REGION Network 109: Step[730] : Z1, Z2 aviod Pos move
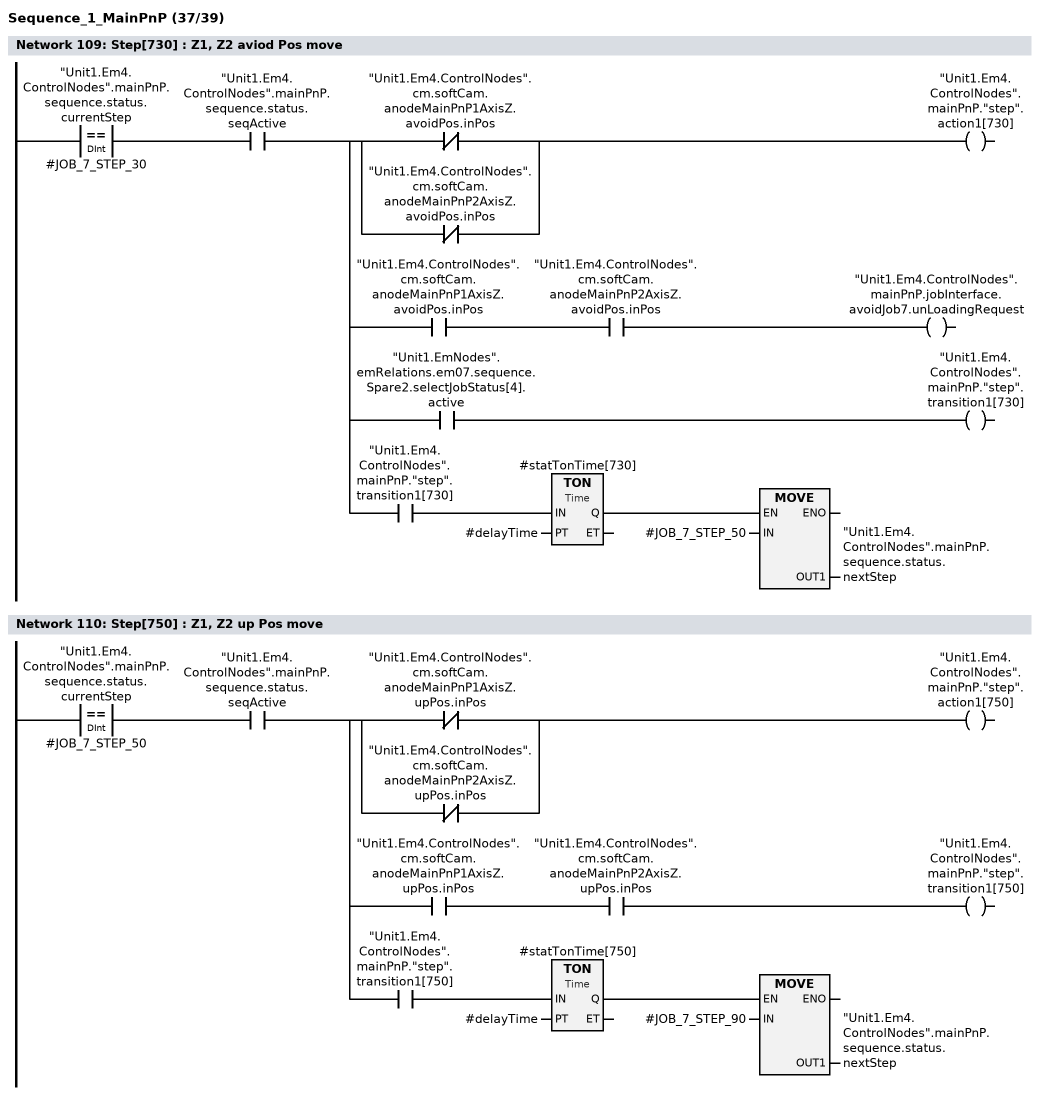
   RUNG wire#powerrail
      { S7_Templates := "SrcType := DInt" } EQ_Contact(in1 := "Unit1.Em4.ControlNodes".mainPnP.sequence.status.currentStep, in2 := #JOB_7_STEP_30)
      Contact( "Unit1.Em4.ControlNodes".mainPnP.sequence.status.seqActive )
      wire#w1
      I_Contact( "Unit1.Em4.ControlNodes".cm.softCam.anodeMainPnP1AxisZ.avoidPos.inPos )
      wire#w2
      Coil( "Unit1.Em4.ControlNodes".mainPnP."step".action1[730] )
   END_RUNG
   RUNG wire#w1
      I_Contact( "Unit1.Em4.ControlNodes".cm.softCam.anodeMainPnP2AxisZ.avoidPos.inPos )
   END_RUNG wire#w2
   RUNG wire#w1
      Contact( "Unit1.Em4.ControlNodes".cm.softCam.anodeMainPnP1AxisZ.avoidPos.inPos )
      Contact( "Unit1.Em4.ControlNodes".cm.softCam.anodeMainPnP2AxisZ.avoidPos.inPos )
      Coil( "Unit1.Em4.ControlNodes".mainPnP.jobInterface.avoidJob7.unLoadingRequest )
   END_RUNG
   RUNG wire#w1
      Contact( "Unit1.EmNodes".emRelations.em07.sequence.Spare2.selectJobStatus[4].active )
      Coil( "Unit1.Em4.ControlNodes".mainPnP."step".transition1[730] )
   END_RUNG
   RUNG wire#w1
      Contact( "Unit1.Em4.ControlNodes".mainPnP."step".transition1[730] )
      { S7_Templates := "time_type := Time" } #statTonTime[730].TON(pt := #delayTime, et =>)
      Move(in := #JOB_7_STEP_50, out1 => "Unit1.Em4.ControlNodes".mainPnP.sequence.status.nextStep)
   END_RUNG
   // the same network as SCL:
   #_w1 := ("Unit1.Em4.ControlNodes".mainPnP.sequence.status.currentStep = #JOB_7_STEP_30) AND "Unit1.Em4.ControlNodes".mainPnP.sequence.status.seqActive;
   "Unit1.Em4.ControlNodes".mainPnP."step".action1[730] := #_w1 AND (NOT "Unit1.Em4.ControlNodes".cm.softCam.anodeMainPnP1AxisZ.avoidPos.inPos OR NOT "Unit1.Em4.ControlNodes".cm.softCam.anodeMainPnP2AxisZ.avoidPos.inPos);
   "Unit1.Em4.ControlNodes".mainPnP.jobInterface.avoidJob7.unLoadingRequest := #_w1 AND "Unit1.Em4.ControlNodes".cm.softCam.anodeMainPnP1AxisZ.avoidPos.inPos AND "Unit1.Em4.ControlNodes".cm.softCam.anodeMainPnP2AxisZ.avoidPos.inPos;
   "Unit1.Em4.ControlNodes".mainPnP."step".transition1[730] := #_w1 AND "Unit1.EmNodes".emRelations.em07.sequence.Spare2.selectJobStatus[4].active;
   #statTonTime[730].TON(IN := #_w1 AND "Unit1.Em4.ControlNodes".mainPnP."step".transition1[730],
                         PT := #delayTime);
   IF #statTonTime[730].Q THEN
       "Unit1.Em4.ControlNodes".mainPnP.sequence.status.nextStep := #JOB_7_STEP_50;
   END_IF;
END_REGION

REGION Network 110: Step[750] : Z1, Z2 up Pos move
   RUNG wire#powerrail
      { S7_Templates := "SrcType := DInt" } EQ_Contact(in1 := "Unit1.Em4.ControlNodes".mainPnP.sequence.status.currentStep, in2 := #JOB_7_STEP_50)
      Contact( "Unit1.Em4.ControlNodes".mainPnP.sequence.status.seqActive )
      wire#w1
      I_Contact( "Unit1.Em4.ControlNodes".cm.softCam.anodeMainPnP1AxisZ.upPos.inPos )
      wire#w2
      Coil( "Unit1.Em4.ControlNodes".mainPnP."step".action1[750] )
   END_RUNG
   RUNG wire#w1
      I_Contact( "Unit1.Em4.ControlNodes".cm.softCam.anodeMainPnP2AxisZ.upPos.inPos )
   END_RUNG wire#w2
   RUNG wire#w1
      Contact( "Unit1.Em4.ControlNodes".cm.softCam.anodeMainPnP1AxisZ.upPos.inPos )
      Contact( "Unit1.Em4.ControlNodes".cm.softCam.anodeMainPnP2AxisZ.upPos.inPos )
      Coil( "Unit1.Em4.ControlNodes".mainPnP."step".transition1[750] )
   END_RUNG
   RUNG wire#w1
      Contact( "Unit1.Em4.ControlNodes".mainPnP."step".transition1[750] )
      { S7_Templates := "time_type := Time" } #statTonTime[750].TON(pt := #delayTime, et =>)
      Move(in := #JOB_7_STEP_90, out1 => "Unit1.Em4.ControlNodes".mainPnP.sequence.status.nextStep)
   END_RUNG
   // the same network as SCL:
   #_w1 := ("Unit1.Em4.ControlNodes".mainPnP.sequence.status.currentStep = #JOB_7_STEP_50) AND "Unit1.Em4.ControlNodes".mainPnP.sequence.status.seqActive;
   "Unit1.Em4.ControlNodes".mainPnP."step".action1[750] := #_w1 AND (NOT "Unit1.Em4.ControlNodes".cm.softCam.anodeMainPnP1AxisZ.upPos.inPos OR NOT "Unit1.Em4.ControlNodes".cm.softCam.anodeMainPnP2AxisZ.upPos.inPos);
   "Unit1.Em4.ControlNodes".mainPnP."step".transition1[750] := #_w1 AND "Unit1.Em4.ControlNodes".cm.softCam.anodeMainPnP1AxisZ.upPos.inPos AND "Unit1.Em4.ControlNodes".cm.softCam.anodeMainPnP2AxisZ.upPos.inPos;
   #statTonTime[750].TON(IN := #_w1 AND "Unit1.Em4.ControlNodes".mainPnP."step".transition1[750],
                         PT := #delayTime);
   IF #statTonTime[750].Q THEN
       "Unit1.Em4.ControlNodes".mainPnP.sequence.status.nextStep := #JOB_7_STEP_90;
   END_IF;
END_REGION

REGION Network 111: Step[790] : JOB[7] Condition
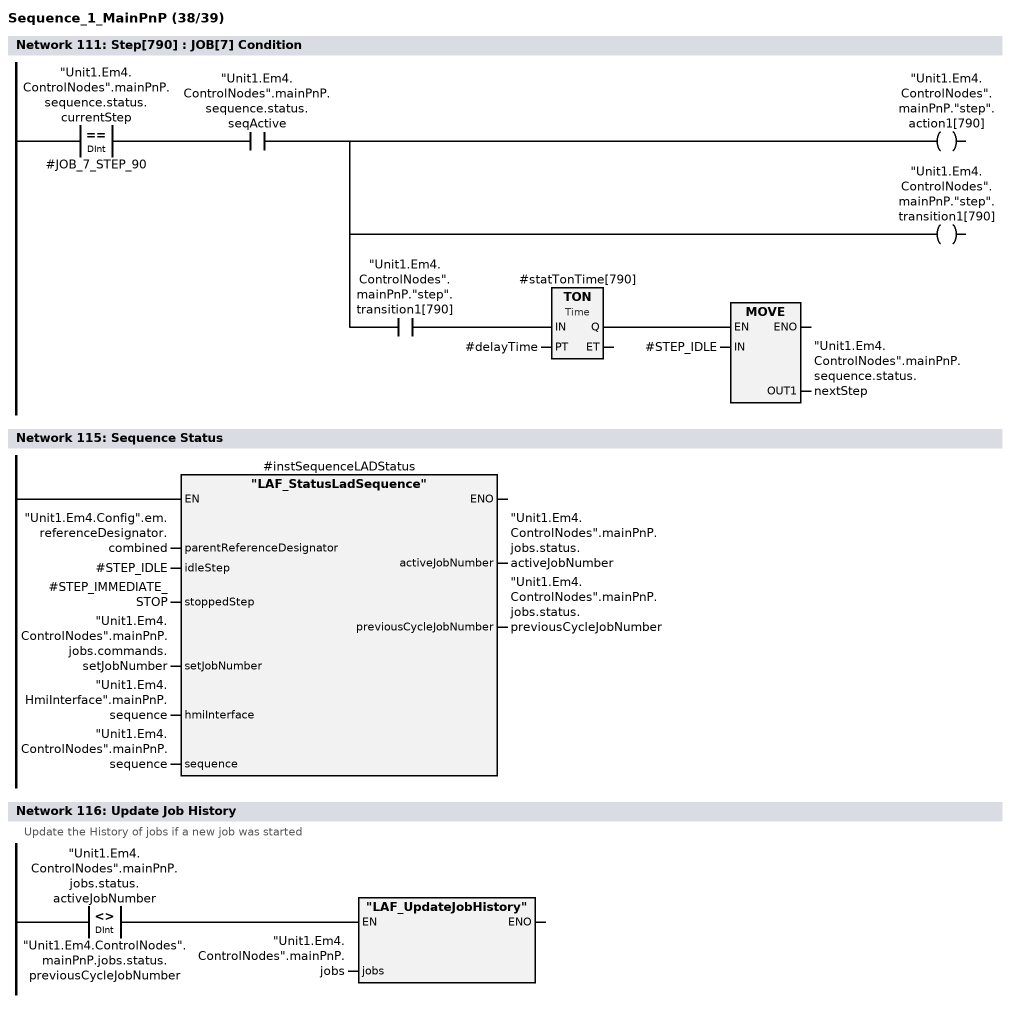
   RUNG wire#powerrail
      { S7_Templates := "SrcType := DInt" } EQ_Contact(in1 := "Unit1.Em4.ControlNodes".mainPnP.sequence.status.currentStep, in2 := #JOB_7_STEP_90)
      Contact( "Unit1.Em4.ControlNodes".mainPnP.sequence.status.seqActive )
      wire#w1
      Coil( "Unit1.Em4.ControlNodes".mainPnP."step".action1[790] )
   END_RUNG
   RUNG wire#w1
      Coil( "Unit1.Em4.ControlNodes".mainPnP."step".transition1[790] )
   END_RUNG
   RUNG wire#w1
      Contact( "Unit1.Em4.ControlNodes".mainPnP."step".transition1[790] )
      { S7_Templates := "time_type := Time" } #statTonTime[790].TON(pt := #delayTime, et =>)
      Move(in := #STEP_IDLE, out1 => "Unit1.Em4.ControlNodes".mainPnP.sequence.status.nextStep)
   END_RUNG
   // the same network as SCL:
   "Unit1.Em4.ControlNodes".mainPnP."step".action1[790] := ("Unit1.Em4.ControlNodes".mainPnP.sequence.status.currentStep = #JOB_7_STEP_90) AND "Unit1.Em4.ControlNodes".mainPnP.sequence.status.seqActive;
   "Unit1.Em4.ControlNodes".mainPnP."step".transition1[790] := ("Unit1.Em4.ControlNodes".mainPnP.sequence.status.currentStep = #JOB_7_STEP_90) AND "Unit1.Em4.ControlNodes".mainPnP.sequence.status.seqActive;
   #statTonTime[790].TON(IN := ("Unit1.Em4.ControlNodes".mainPnP.sequence.status.currentStep = #JOB_7_STEP_90) AND "Unit1.Em4.ControlNodes".mainPnP.sequence.status.seqActive AND "Unit1.Em4.ControlNodes".mainPnP."step".transition1[790],
                         PT := #delayTime);
   IF #statTonTime[790].Q THEN
       "Unit1.Em4.ControlNodes".mainPnP.sequence.status.nextStep := #STEP_IDLE;
   END_IF;
END_REGION

REGION Network 112: *************** IMMEDIATE STOP **************************
END_REGION

REGION Network 113: Immediate Stop
END_REGION

REGION Network 114: *************** Status updates **************************
END_REGION

REGION Network 115: Sequence Status
   RUNG wire#powerrail
      #instSequenceLADStatus(parentReferenceDesignator := "Unit1.Em4.Config".em.referenceDesignator.combined, idleStep := #STEP_IDLE, stoppedStep := #STEP_IMMEDIATE_STOP, setJobNumber := "Unit1.Em4.ControlNodes".mainPnP.jobs.commands.setJobNumber, hmiInterface := "Unit1.Em4.HmiInterface".mainPnP.sequence, sequence := "Unit1.Em4.ControlNodes".mainPnP.sequence, activeJobNumber => "Unit1.Em4.ControlNodes".mainPnP.jobs.status.activeJobNumber, previousCycleJobNumber => "Unit1.Em4.ControlNodes".mainPnP.jobs.status.previousCycleJobNumber)
   END_RUNG
   // the same network as SCL:
   #instSequenceLADStatus(parentReferenceDesignator := "Unit1.Em4.Config".em.referenceDesignator.combined,   // "LAF_StatusLadSequence"
                          idleStep := #STEP_IDLE,
                          stoppedStep := #STEP_IMMEDIATE_STOP,
                          setJobNumber := "Unit1.Em4.ControlNodes".mainPnP.jobs.commands.setJobNumber,
                          hmiInterface := "Unit1.Em4.HmiInterface".mainPnP.sequence,
                          sequence := "Unit1.Em4.ControlNodes".mainPnP.sequence,
                          activeJobNumber => "Unit1.Em4.ControlNodes".mainPnP.jobs.status.activeJobNumber,
                          previousCycleJobNumber => "Unit1.Em4.ControlNodes".mainPnP.jobs.status.previousCycleJobNumber);
END_REGION

REGION Network 116: Update Job History
   // Update the History of jobs if a new job was started
   RUNG wire#powerrail
      { S7_Templates := "SrcType := DInt" } NE_Contact(in1 := "Unit1.Em4.ControlNodes".mainPnP.jobs.status.activeJobNumber, in2 := "Unit1.Em4.ControlNodes".mainPnP.jobs.status.previousCycleJobNumber)
      "LAF_UpdateJobHistory"(jobs := "Unit1.Em4.ControlNodes".mainPnP.jobs)
   END_RUNG
   // the same network as SCL:
   IF "Unit1.Em4.ControlNodes".mainPnP.jobs.status.activeJobNumber <> "Unit1.Em4.ControlNodes".mainPnP.jobs.status.previousCycleJobNumber THEN
       "LAF_UpdateJobHistory"(jobs := "Unit1.Em4.ControlNodes".mainPnP.jobs);
   END_IF;
END_REGION

REGION Network 117: Output steps as String
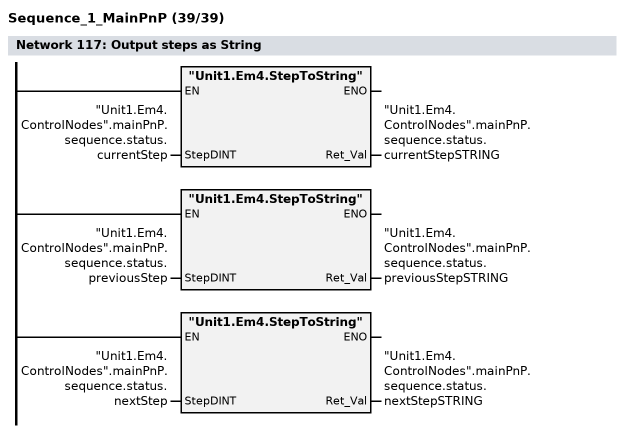
   RUNG wire#powerrail
      "Unit1.Em4.StepToString"(StepDINT := "Unit1.Em4.ControlNodes".mainPnP.sequence.status.currentStep, Ret_Val => "Unit1.Em4.ControlNodes".mainPnP.sequence.status.currentStepSTRING)
   END_RUNG
   RUNG wire#powerrail
      "Unit1.Em4.StepToString"(StepDINT := "Unit1.Em4.ControlNodes".mainPnP.sequence.status.previousStep, Ret_Val => "Unit1.Em4.ControlNodes".mainPnP.sequence.status.previousStepSTRING)
   END_RUNG
   RUNG wire#powerrail
      "Unit1.Em4.StepToString"(StepDINT := "Unit1.Em4.ControlNodes".mainPnP.sequence.status.nextStep, Ret_Val => "Unit1.Em4.ControlNodes".mainPnP.sequence.status.nextStepSTRING)
   END_RUNG
   // the same network as SCL:
   "Unit1.Em4.ControlNodes".mainPnP.sequence.status.currentStepSTRING := "Unit1.Em4.StepToString"(StepDINT := "Unit1.Em4.ControlNodes".mainPnP.sequence.status.currentStep);
   "Unit1.Em4.ControlNodes".mainPnP.sequence.status.previousStepSTRING := "Unit1.Em4.StepToString"(StepDINT := "Unit1.Em4.ControlNodes".mainPnP.sequence.status.previousStep);
   "Unit1.Em4.ControlNodes".mainPnP.sequence.status.nextStepSTRING := "Unit1.Em4.StepToString"(StepDINT := "Unit1.Em4.ControlNodes".mainPnP.sequence.status.nextStep);
END_REGION
END_FUNCTION_BLOCK
